PROGRAM OpenFremwork_TestRunner
VAR
	testAutomationUnit : TestAutomationUnit;
	automationUnits : ARRAY [0..0] OF AutomationEngine.IAutomationUnit := [testAutomationUnit];
	
	automationRunner :  AutomationEngine.AutomationRunner;
END_VAR

automationRunner.Run(automationUnits);

END_PROGRAM

(* stored: Version 1.1.0.1, ProductVersion 3.1.4026.12
   POU OpenFremwork_TestRunner: Id {e4eb2eaa-3c4c-0200-2bd5-f94fd2ee20dd}, SpecialFunc None *)
